FUNCTION_BLOCK FB_SLIDERL (* FB_SLIDER with local publication of position *)
  (* Standard: 61499-1; Classification: HMI *)
  (* Version 0.0, 2006-11-03, JHC, Holobloc Inc, Copied/Modified from MECH_HMIL. *)
  (* Compiler header: package fb.rt.hmi; import fb.rt.mva.FBMVCD; import fb.rt.net.*; *)
  (* Compiler classdef: public class FB_SLIDERL extends FBMVCD *)
  (* Compiler Java Sun JDK 1.5.0 *)
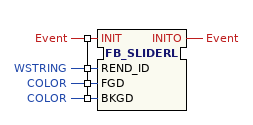
  EVENT_INPUT
    INIT WITH REND_ID, BKGD, FGD; (* Initialization Request *)
  END_EVENT
  EVENT_OUTPUT
    INITO; (* Initialization Confirm *)
  END_EVENT
  VAR_INPUT
    REND_ID : WSTRING; (* Data Channel ID - default is FB instaqnce name *)
    FGD : COLOR := red; (* Slider Foreground Color *)
    BKGD : COLOR := blue; (* Slider Background Color *)
  END_VAR
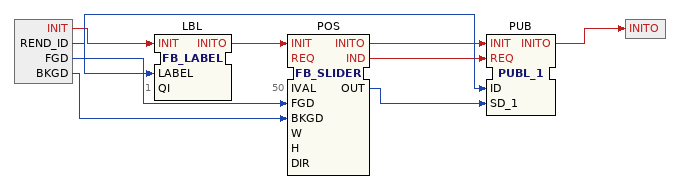
  FBS
    LBL : FB_LABEL(QI := 1);
    POS : FB_SLIDER(IVAL := 50);
    PUB : PUBL_1;
  END_FBS
  EVENT_CONNECTIONS
    INIT TO LBL.INIT;
    LBL.INITO TO POS.INIT;
    PUB.INITO TO INITO;
    POS.INITO TO PUB.INIT;
    POS.IND TO PUB.REQ;
  END_CONNECTIONS
  DATA_CONNECTIONS
    REND_ID TO PUB.ID;
    REND_ID TO LBL.LABEL;
    POS.OUT TO PUB.SD_1;
    FGD TO POS.FGD;
    BKGD TO POS.BKGD;
  END_CONNECTIONS
END_FUNCTION_BLOCK
